(* IEC 61131-3 sources: AXOpen/src/template.axolibrary/app/src, 2 files *)

(* ---- configuration.st ---- *)
USING Template.Axolibrary;

CONFIGURATION MyConfiguration
    TASK Main(Interval := T#10ms, Priority := 1);
    PROGRAM P1 WITH Main: MyProgram;

    VAR_GLOBAL
        {S7.extern=ReadWrite}
        sandbox : Template.Axolibrary.SandboxContext;
        {S7.extern=ReadWrite}
        documentation : Template.Axolibrary.DocumentationContext;
        {S7.extern=ReadWrite}
        _rtc : AXOpen.S71500.Rtc;
        {S7.extern=ReadWrite}
        _rtm : AXOpen.S71500.Rtm;
    END_VAR

END_CONFIGURATION

(* ---- program.st ---- *)
USING Template.Axolibrary;

PROGRAM MyProgram
    VAR_EXTERNAL
        sandbox : Template.Axolibrary.SandboxContext;
        documentation : Template.Axolibrary.DocumentationContext;
        _rtc : AXOpen.S71500.Rtc;
        _rtm : AXOpen.S71500.Rtm;
    END_VAR

    sandbox.InjectRtc(_rtc);
    sandbox.InjectRtm(_rtm);
    sandbox.Run();

    documentation.InjectRtc(_rtc);
    documentation.InjectRtm(_rtm);
    documentation.Run();
END_PROGRAM
